LIN {X 0,Y 119.438,Z 237.503,A -85,B 0,C 180,E1 -30793.611,E2 -30793.611} C_VEL
LIN {X 0,Y 118.662,Z 241.868,A -85,B 0,C 180,E1 -30795.896,E2 -30795.896} C_VEL
LIN {X 0,Y 115.868,Z 252.745,A -85,B 0,C 180,E1 -30800.631,E2 -30800.631} C_VEL
LIN {X 0,Y 112.821,Z 263.888,A -85,B 0,C 180,E1 -30806.572,E2 -30806.572} C_VEL
LIN {X 0,Y 111.137,Z 271.247,A -85,B 0,C 180,E1 -30811.379,E2 -30811.379} C_VEL
LIN {X 0,Y 110.077,Z 278.124,A -85,B 0,C 180,E1 -30816.678,E2 -30816.678} C_VEL
LIN {X 0,Y 109.957,Z 285.411,A -85,B 0,C 180,E1 -30823.396,E2 -30823.396} C_VEL
LIN {X 0,Y 111.695,Z 292.264,A -85,B 0,C 180,E1 -30831.008,E2 -30831.008} C_VEL
LIN {X 0,Y 115.498,Z 297.926,A -85,B 0,C 180,E1 -30838.414,E2 -30838.414} C_VEL
LIN {X 0,Y 120.449,Z 301.979,A -85,B 0,C 180,E1 -30844.487,E2 -30844.487} C_VEL
LIN {X 0,Y 127.678,Z 305.592,A -85,B 0,C 180,E1 -30850.715,E2 -30850.715} C_VEL
LIN {X 0,Y 137.267,Z 308.443,A -85,B 0,C 180,E1 -30856.596,E2 -30856.596} C_VEL
LIN {X 0,Y 149.082,Z 310.385,A -85,B 0,C 180,E1 -30861.87,E2 -30861.87} C_VEL
LIN {X 0,Y 161.99,Z 311.348,A -85,B 0,C 180,E1 -30866.234,E2 -30866.234} C_VEL
LIN {X 0,Y 176.136,Z 311.421,A -85,B 0,C 180,E1 -30870,E2 -30870} C_VEL
LIN {X 0,Y 161.989,Z 311.349,A -85,B 0,C 180,E1 -30873.762,E2 -30873.762} C_VEL
LIN {X 0,Y 158.576,Z 311.223,A -85,B 0,C 180,E1 -30874.811,E2 -30874.811} C_VEL
LIN {X 0,Y 153.772,Z 311.084,A -85,B 0,C 180,E1 -30876.072,E2 -30876.072} C_VEL
LIN {X 0,Y 137.981,Z 310.516,A -85,B 0,C 180,E1 -30879.329,E2 -30879.329} C_VEL
LIN {X 0,Y 132.654,Z 310.062,A -85,B 0,C 180,E1 -30881.151,E2 -30881.151} C_VEL
LIN {X 0,Y 132.002,Z 309.878,A -85,B 0,C 180,E1 -30881.466,E2 -30881.466} C_VEL
LIN {X 0,Y 123.49,Z 307.999,A -85,B 0,C 180,E1 -30886.532,E2 -30886.532} C_VEL
LIN {X 0,Y 114.976,Z 304.68,A -85,B 0,C 180,E1 -30893.529,E2 -30893.529} C_VEL
LIN {X 0,Y 108.155,Z 299.529,A -85,B 0,C 180,E1 -30902.359,E2 -30902.359} C_VEL
LIN {X 0,Y 104.971,Z 294.579,A -85,B 0,C 180,E1 -30909.654,E2 -30909.654} C_VEL
LIN {X 0,Y 103.68,Z 288.412,A -85,B 0,C 180,E1 -30917.327,E2 -30917.327} C_VEL
LIN {X 0,Y 103.938,Z 283.545,A -85,B 0,C 180,E1 -30922.518,E2 -30922.518} C_VEL
LIN {X 0,Y 105.318,Z 276.622,A -85,B 0,C 180,E1 -30928.735,E2 -30928.735} C_VEL
LIN {X 0,Y 107.837,Z 268.159,A -85,B 0,C 180,E1 -30934.941,E2 -30934.941} C_VEL
LIN {X 0,Y 110.814,Z 259.529,A -85,B 0,C 180,E1 -30940.073,E2 -30940.073} C_VEL
LIN {X 0,Y 113.576,Z 251.659,A -85,B 0,C 180,E1 -30943.971,E2 -30943.971} C_VEL
LIN {X 0,Y 115.588,Z 245.687,A -85,B 0,C 180,E1 -30946.614,E2 -30946.614} C_VEL
LIN {X 0,Y 116.453,Z 242.049,A -85,B 0,C 180,E1 -30948.603,E2 -30948.603} C_VEL
LIN {X 0,Y 117.198,Z 238.265,A -85,B 0,C 180,E1 -30951.38,E2 -30951.38} C_VEL
LIN {X 0,Y 117.648,Z 235.676,A -85,B 0,C 180,E1 -30954.17,E2 -30954.17} C_VEL
LIN {X 0,Y 117.803,Z 234.235,A -85,B 0,C 180,E1 -30956.582,E2 -30956.582} C_VEL
LIN {X 0,Y 118.145,Z 232.807,A -85,B 0,C 180,E1 -30960.002,E2 -30960.002} C_VEL
LIN {X 0,Y 117.857,Z 233.676,A -85,B 0,C 180,E1 -30960.329,E2 -30960.329} C_VEL
LIN {X 0,Y 112.453,Z 246.435,A -85,B 0,C 180,E1 -30960.571,E2 -30960.571} C_VEL
LIN {X 0,Y 106.312,Z 257.337,A -85,B 0,C 180,E1 -30960.916,E2 -30960.916} C_VEL
LIN {X 0,Y 100.174,Z 266.275,A -85,B 0,C 180,E1 -30961.292,E2 -30961.292} C_VEL
LIN {X 0,Y 93.166,Z 274.795,A -85,B 0,C 180,E1 -30961.794,E2 -30961.794} C_VEL
LIN {X 0,Y 86.168,Z 282.007,A -85,B 0,C 180,E1 -30962.392,E2 -30962.392} C_VEL
LIN {X 0,Y 79.184,Z 288.203,A -85,B 0,C 180,E1 -30963.148,E2 -30963.148} C_VEL
LIN {X 0,Y 70.479,Z 294.736,A -85,B 0,C 180,E1 -30964.311,E2 -30964.311} C_VEL
LIN {X 0,Y 63.549,Z 299.237,A -85,B 0,C 180,E1 -30965.543,E2 -30965.543} C_VEL
LIN {X 0,Y 52.229,Z 305.189,A -85,B 0,C 180,E1 -30968.35,E2 -30968.35} C_VEL
LIN {X 0,Y 43.035,Z 309.057,A -85,B 0,C 180,E1 -30971.523,E2 -30971.523} C_VEL
LIN {X 0,Y 36.377,Z 311.428,A -85,B 0,C 180,E1 -30974.988,E2 -30974.988} C_VEL
LIN {X 0,Y 29.876,Z 313.231,A -85,B 0,C 180,E1 -30979.79,E2 -30979.79} C_VEL
LIN {X 0,Y 18.303,Z 315.698,A -85,B 0,C 180,E1 -30999.83,E2 -30999.83} C_VEL
LIN {X 0,Y 14.254,Z 316.299,A -85,B 0,C 180,E1 -31020.458,E2 -31020.458} C_VEL
LIN {X 0,Y 12.863,Z 316.464,A -85,B 0,C 180,E1 -31050,E2 -31050} C_VEL
LIN {X 0,Y 14.212,Z 316.298,A -85,B 0,C 180,E1 -31079.637,E2 -31079.637} C_VEL
LIN {X 0,Y 18.3,Z 315.698,A -85,B 0,C 180,E1 -31100.182,E2 -31100.182} C_VEL
LIN {X 0,Y 29.876,Z 313.231,A -85,B 0,C 180,E1 -31120.21,E2 -31120.21} C_VEL
LIN {X 0,Y 39.696,Z 310.276,A -85,B 0,C 180,E1 -31126.842,E2 -31126.842} C_VEL
LIN {X 0,Y 49.826,Z 306.286,A -85,B 0,C 180,E1 -31130.878,E2 -31130.878} C_VEL
LIN {X 0,Y 56.662,Z 303.07,A -85,B 0,C 180,E1 -31132.871,E2 -31132.871} C_VEL
LIN {X 0,Y 67.011,Z 297.047,A -85,B 0,C 180,E1 -31135.094,E2 -31135.094} C_VEL
LIN {X 0,Y 75.7,Z 290.954,A -85,B 0,C 180,E1 -31136.406,E2 -31136.406} C_VEL
LIN {X 0,Y 82.676,Z 285.259,A -85,B 0,C 180,E1 -31137.218,E2 -31137.218} C_VEL
LIN {X 0,Y 91.415,Z 276.712,A -85,B 0,C 180,E1 -31138.075,E2 -31138.075} C_VEL
LIN {X 0,Y 98.421,Z 268.542,A -85,B 0,C 180,E1 -31138.594,E2 -31138.594} C_VEL
LIN {X 0,Y 104.558,Z 260.038,A -85,B 0,C 180,E1 -31138.98,E2 -31138.98} C_VEL
LIN {X 0,Y 109.821,Z 251.33,A -85,B 0,C 180,E1 -31139.273,E2 -31139.273} C_VEL
LIN {X 0,Y 114.56,Z 241.781,A -85,B 0,C 180,E1 -31139.51,E2 -31139.51} C_VEL
LIN {X 0,Y 117.857,Z 233.673,A -85,B 0,C 180,E1 -31139.689,E2 -31139.689} C_VEL
LIN {X 0,Y 118.131,Z 232.849,A -85,B 0,C 180,E1 -31139.998,E2 -31139.998} C_VEL
LIN {X 0,Y 117.796,Z 234.256,A -85,B 0,C 180,E1 -31143.419,E2 -31143.419} C_VEL
LIN {X 0,Y 117.508,Z 236.547,A -85,B 0,C 180,E1 -31146.868,E2 -31146.868} C_VEL
LIN {X 0,Y 116.994,Z 239.333,A -85,B 0,C 180,E1 -31149.507,E2 -31149.507} C_VEL
LIN {X 0,Y 116.087,Z 243.786,A -85,B 0,C 180,E1 -31152.409,E2 -31152.409} C_VEL
LIN {X 0,Y 114.525,Z 248.785,A -85,B 0,C 180,E1 -31154.767,E2 -31154.767} C_VEL
LIN {X 0,Y 111.471,Z 257.668,A -85,B 0,C 180,E1 -31158.966,E2 -31158.966} C_VEL
LIN {X 0,Y 109.077,Z 264.504,A -85,B 0,C 180,E1 -31162.74,E2 -31162.74} C_VEL
LIN {X 0,Y 106.284,Z 272.99,A -85,B 0,C 180,E1 -31168.437,E2 -31168.437} C_VEL
LIN {X 0,Y 104.433,Z 280.285,A -85,B 0,C 180,E1 -31174.431,E2 -31174.431} C_VEL
LIN {X 0,Y 103.677,Z 286.441,A -85,B 0,C 180,E1 -31180.481,E2 -31180.481} C_VEL
LIN {X 0,Y 104.336,Z 292.655,A -85,B 0,C 180,E1 -31187.809,E2 -31187.809} C_VEL
LIN {X 0,Y 106.867,Z 298.01,A -85,B 0,C 180,E1 -31195.284,E2 -31195.284} C_VEL
LIN {X 0,Y 111.215,Z 302.267,A -85,B 0,C 180,E1 -31202.21,E2 -31202.21} C_VEL
LIN {X 0,Y 117.696,Z 305.878,A -85,B 0,C 180,E1 -31209.006,E2 -31209.006} C_VEL
LIN {X 0,Y 124.268,Z 308.213,A -85,B 0,C 180,E1 -31214.031,E2 -31214.031} C_VEL
LIN {X 0,Y 135.497,Z 310.434,A -85,B 0,C 180,E1 -31220.219,E2 -31220.219} C_VEL
LIN {X 0,Y 148.094,Z 311.583,A -85,B 0,C 180,E1 -31225.244,E2 -31225.244} C_VEL
LIN {X 0,Y 164.15,Z 311.737,A -85,B 0,C 180,E1 -31230,E2 -31230} C_VEL
LIN {X 0,Y 148.093,Z 311.584,A -85,B 0,C 180,E1 -31234.753,E2 -31234.753} C_VEL
LIN {X 0,Y 135.49,Z 310.441,A -85,B 0,C 180,E1 -31239.764,E2 -31239.764} C_VEL
LIN {X 0,Y 132.002,Z 309.878,A -85,B 0,C 180,E1 -31241.466,E2 -31241.466} C_VEL
LIN {X 0,Y 127.809,Z 309.35,A -85,B 0,C 180,E1 -31243.289,E2 -31243.289} C_VEL
LIN {X 0,Y 113.917,Z 307.957,A -85,B 0,C 180,E1 -31248.551,E2 -31248.551} C_VEL
LIN {X 0,Y 110.162,Z 307.095,A -85,B 0,C 180,E1 -31250.829,E2 -31250.829} C_VEL
LIN {X 0,Y 109.172,Z 306.728,A -85,B 0,C 180,E1 -31251.693,E2 -31251.693} C_VEL
LIN {X 0,Y 103.628,Z 303.627,A -85,B 0,C 180,E1 -31258.342,E2 -31258.342} C_VEL
LIN {X 0,Y 99.465,Z 299.348,A -85,B 0,C 180,E1 -31266.219,E2 -31266.219} C_VEL
LIN {X 0,Y 97.579,Z 294.398,A -85,B 0,C 180,E1 -31273.929,E2 -31273.929} C_VEL
LIN {X 0,Y 97.658,Z 287.855,A -85,B 0,C 180,E1 -31282.337,E2 -31282.337} C_VEL
LIN {X 0,Y 99.07,Z 282.136,A -85,B 0,C 180,E1 -31288.35,E2 -31288.35} C_VEL
LIN {X 0,Y 101.484,Z 275.444,A -85,B 0,C 180,E1 -31294.195,E2 -31294.195} C_VEL
LIN {X 0,Y 104.802,Z 267.508,A -85,B 0,C 180,E1 -31299.857,E2 -31299.857} C_VEL
LIN {X 0,Y 108.121,Z 259.958,A -85,B 0,C 180,E1 -31304.221,E2 -31304.221} C_VEL
LIN {X 0,Y 111.79,Z 251.291,A -85,B 0,C 180,E1 -31308.348,E2 -31308.348} C_VEL
LIN {X 0,Y 113.189,Z 247.517,A -85,B 0,C 180,E1 -31310.304,E2 -31310.304} C_VEL
LIN {X 0,Y 114.31,Z 243.924,A -85,B 0,C 180,E1 -31312.939,E2 -31312.939} C_VEL
LIN {X 0,Y 114.701,Z 242.248,A -85,B 0,C 180,E1 -31314.729,E2 -31314.729} C_VEL
LIN {X 0,Y 114.969,Z 241.111,A -85,B 0,C 180,E1 -31316.497,E2 -31316.497} C_VEL
LIN {X 0,Y 114.315,Z 242.512,A -85,B 0,C 180,E1 -31316.943,E2 -31316.943} C_VEL
LIN {X 0,Y 108.197,Z 254.379,A -85,B 0,C 180,E1 -31317.066,E2 -31317.066} C_VEL
LIN {X 0,Y 101.147,Z 264.951,A -85,B 0,C 180,E1 -31317.212,E2 -31317.212} C_VEL
LIN {X 0,Y 94.979,Z 272.687,A -85,B 0,C 180,E1 -31317.355,E2 -31317.355} C_VEL
LIN {X 0,Y 86.165,Z 281.815,A -85,B 0,C 180,E1 -31317.655,E2 -31317.655} C_VEL
LIN {X 0,Y 79.113,Z 288.012,A -85,B 0,C 180,E1 -31317.99,E2 -31317.99} C_VEL
LIN {X 0,Y 70.303,Z 294.545,A -85,B 0,C 180,E1 -31318.526,E2 -31318.526} C_VEL
LIN {X 0,Y 63.26,Z 299.045,A -85,B 0,C 180,E1 -31319.081,E2 -31319.081} C_VEL
LIN {X 0,Y 53.186,Z 304.328,A -85,B 0,C 180,E1 -31320.252,E2 -31320.252} C_VEL
LIN {X 0,Y 42.194,Z 308.865,A -85,B 0,C 180,E1 -31322.001,E2 -31322.001} C_VEL
LIN {X 0,Y 35.214,Z 311.237,A -85,B 0,C 180,E1 -31323.728,E2 -31323.728} C_VEL
LIN {X 0,Y 28.271,Z 313.04,A -85,B 0,C 180,E1 -31326.077,E2 -31326.077} C_VEL
LIN {X 0,Y 14.788,Z 315.507,A -85,B 0,C 180,E1 -31338.102,E2 -31338.102} C_VEL
LIN {X 0,Y 8.796,Z 316.109,A -85,B 0,C 180,E1 -31356.968,E2 -31356.968} C_VEL
LIN {X 0,Y 5.75,Z 316.273,A -85,B 0,C 180,E1 -31410,E2 -31410} C_VEL
LIN {X 0,Y 8.773,Z 316.108,A -85,B 0,C 180,E1 -31463.232,E2 -31463.232} C_VEL
LIN {X 0,Y 14.787,Z 315.507,A -85,B 0,C 180,E1 -31481.914,E2 -31481.914} C_VEL
LIN {X 0,Y 28.271,Z 313.04,A -85,B 0,C 180,E1 -31493.923,E2 -31493.923} C_VEL
LIN {X 0,Y 38.7,Z 310.085,A -85,B 0,C 180,E1 -31497.19,E2 -31497.19} C_VEL
LIN {X 0,Y 49.202,Z 306.095,A -85,B 0,C 180,E1 -31499.114,E2 -31499.114} C_VEL
LIN {X 0,Y 56.224,Z 302.878,A -85,B 0,C 180,E1 -31500.109,E2 -31500.109} C_VEL
LIN {X 0,Y 66.78,Z 296.856,A -85,B 0,C 180,E1 -31501.191,E2 -31501.191} C_VEL
LIN {X 0,Y 75.588,Z 290.762,A -85,B 0,C 180,E1 -31501.807,E2 -31501.807} C_VEL
LIN {X 0,Y 82.636,Z 285.068,A -85,B 0,C 180,E1 -31502.141,E2 -31502.141} C_VEL
LIN {X 0,Y 91.452,Z 276.521,A -85,B 0,C 180,E1 -31502.524,E2 -31502.524} C_VEL
LIN {X 0,Y 98.503,Z 268.351,A -85,B 0,C 180,E1 -31502.724,E2 -31502.724} C_VEL
LIN {X 0,Y 104.673,Z 259.847,A -85,B 0,C 180,E1 -31502.872,E2 -31502.872} C_VEL
LIN {X 0,Y 110.366,Z 250.392,A -85,B 0,C 180,E1 -31503.004,E2 -31503.004} C_VEL
LIN {X 0,Y 114.153,Z 242.882,A -85,B 0,C 180,E1 -31503.048,E2 -31503.048} C_VEL
LIN {X 0,Y 114.958,Z 241.136,A -85,B 0,C 180,E1 -31503.503,E2 -31503.503} C_VEL
LIN {X 0,Y 114.708,Z 242.232,A -85,B 0,C 180,E1 -31505.271,E2 -31505.271} C_VEL
LIN {X 0,Y 114.078,Z 244.695,A -85,B 0,C 180,E1 -31507.642,E2 -31507.642} C_VEL
LIN {X 0,Y 113.171,Z 247.553,A -85,B 0,C 180,E1 -31509.699,E2 -31509.699} C_VEL
LIN {X 0,Y 111.781,Z 251.303,A -85,B 0,C 180,E1 -31511.648,E2 -31511.648} C_VEL
LIN {X 0,Y 107.546,Z 261.415,A -85,B 0,C 180,E1 -31516.579,E2 -31516.579} C_VEL
LIN {X 0,Y 102.944,Z 271.932,A -85,B 0,C 180,E1 -31523.11,E2 -31523.11} C_VEL
LIN {X 0,Y 99.555,Z 280.572,A -85,B 0,C 180,E1 -31530.147,E2 -31530.147} C_VEL
LIN {X 0,Y 97.91,Z 286.701,A -85,B 0,C 180,E1 -31536.364,E2 -31536.364} C_VEL
LIN {X 0,Y 97.409,Z 292.784,A -85,B 0,C 180,E1 -31543.823,E2 -31543.823} C_VEL
LIN {X 0,Y 98.744,Z 297.982,A -85,B 0,C 180,E1 -31551.524,E2 -31551.524} C_VEL
LIN {X 0,Y 102.104,Z 302.412,A -85,B 0,C 180,E1 -31559.271,E2 -31559.271} C_VEL
LIN {X 0,Y 107.87,Z 306.162,A -85,B 0,C 180,E1 -31566.989,E2 -31566.989} C_VEL
LIN {X 0,Y 113.189,Z 308.289,A -85,B 0,C 180,E1 -31571.914,E2 -31571.914} C_VEL
LIN {X 0,Y 122.122,Z 310.418,A -85,B 0,C 180,E1 -31578.042,E2 -31578.042} C_VEL
LIN {X 0,Y 134.394,Z 311.803,A -85,B 0,C 180,E1 -31583.997,E2 -31583.997} C_VEL
LIN {X 0,Y 147.624,Z 312.173,A -85,B 0,C 180,E1 -31588.66,E2 -31588.66} C_VEL
LIN {X 0,Y 152.223,Z 312.051,A -85,B 0,C 180,E1 -31590,E2 -31590} C_VEL
LIN {X 0,Y 140.825,Z 312.065,A -85,B 0,C 180,E1 -31593.543,E2 -31593.543} C_VEL
LIN {X 0,Y 128.009,Z 311.191,A -85,B 0,C 180,E1 -31598.806,E2 -31598.806} C_VEL
LIN {X 0,Y 119.334,Z 309.848,A -85,B 0,C 180,E1 -31603.625,E2 -31603.625} C_VEL
LIN {X 0,Y 111.719,Z 307.776,A -85,B 0,C 180,E1 -31609.338,E2 -31609.338} C_VEL
LIN {X 0,Y 109.172,Z 306.728,A -85,B 0,C 180,E1 -31611.693,E2 -31611.693} C_VEL
LIN {X 0,Y 106.013,Z 305.743,A -85,B 0,C 180,E1 -31614.302,E2 -31614.302} C_VEL
LIN {X 0,Y 95.36,Z 303.145,A -85,B 0,C 180,E1 -31622.33,E2 -31622.33} C_VEL
LIN {X 0,Y 92.785,Z 301.661,A -85,B 0,C 180,E1 -31626.088,E2 -31626.088} C_VEL
LIN {X 0,Y 92.582,Z 301.332,A -85,B 0,C 180,E1 -31626.657,E2 -31626.657} C_VEL
LIN {X 0,Y 90.988,Z 296.082,A -85,B 0,C 180,E1 -31635.963,E2 -31635.963} C_VEL
LIN {X 0,Y 91.838,Z 289.677,A -85,B 0,C 180,E1 -31644.98,E2 -31644.98} C_VEL
LIN {X 0,Y 94.652,Z 282.378,A -85,B 0,C 180,E1 -31653,E2 -31653} C_VEL
LIN {X 0,Y 98.048,Z 275.499,A -85,B 0,C 180,E1 -31659.001,E2 -31659.001} C_VEL
LIN {X 0,Y 101.83,Z 268.389,A -85,B 0,C 180,E1 -31663.977,E2 -31663.977} C_VEL
LIN {X 0,Y 106.055,Z 260.347,A -85,B 0,C 180,E1 -31668.535,E2 -31668.535} C_VEL
LIN {X 0,Y 109.351,Z 253.877,A -85,B 0,C 180,E1 -31671.616,E2 -31671.616} C_VEL
LIN {X 0,Y 110.135,Z 251.985,A -85,B 0,C 180,E1 -31672.67,E2 -31672.67} C_VEL
LIN {X 0,Y 109.077,Z 253.677,A -85,B 0,C 180,E1 -31673.347,E2 -31673.347} C_VEL
LIN {X 0,Y 101.741,Z 264.76,A -85,B 0,C 180,E1 -31673.207,E2 -31673.207} C_VEL
LIN {X 0,Y 95.568,Z 272.496,A -85,B 0,C 180,E1 -31673.107,E2 -31673.107} C_VEL
LIN {X 0,Y 86.75,Z 281.624,A -85,B 0,C 180,E1 -31672.94,E2 -31672.94} C_VEL
LIN {X 0,Y 79.683,Z 287.821,A -85,B 0,C 180,E1 -31672.859,E2 -31672.859} C_VEL
LIN {X 0,Y 70.846,Z 294.353,A -85,B 0,C 180,E1 -31672.75,E2 -31672.75} C_VEL
LIN {X 0,Y 63.775,Z 298.853,A -85,B 0,C 180,E1 -31672.658,E2 -31672.658} C_VEL
LIN {X 0,Y 52.639,Z 304.573,A -85,B 0,C 180,E1 -31672.585,E2 -31672.585} C_VEL
LIN {X 0,Y 42.544,Z 308.674,A -85,B 0,C 180,E1 -31672.375,E2 -31672.375} C_VEL
LIN {X 0,Y 35.47,Z 311.046,A -85,B 0,C 180,E1 -31672.177,E2 -31672.177} C_VEL
LIN {X 0,Y 28.413,Z 312.849,A -85,B 0,C 180,E1 -31671.655,E2 -31671.655} C_VEL
LIN {X 0,Y 14.285,Z 315.315,A -85,B 0,C 180,E1 -31669.716,E2 -31669.716} C_VEL
LIN {X 0,Y 7.266,Z 315.917,A -85,B 0,C 180,E1 -31665.308,E2 -31665.308} C_VEL
LIN {X 0,Y 1.349,Z 316.083,A -85,B 0,C 180,E1 -31590,E2 -31590} C_VEL
LIN {X 0,Y 7.274,Z 315.916,A -85,B 0,C 180,E1 -31514.942,E2 -31514.942} C_VEL
LIN {X 0,Y 14.286,Z 315.315,A -85,B 0,C 180,E1 -31510.299,E2 -31510.299} C_VEL
LIN {X 0,Y 28.413,Z 312.849,A -85,B 0,C 180,E1 -31508.345,E2 -31508.345} C_VEL
LIN {X 0,Y 39.009,Z 309.893,A -85,B 0,C 180,E1 -31507.738,E2 -31507.738} C_VEL
LIN {X 0,Y 49.608,Z 305.903,A -85,B 0,C 180,E1 -31507.387,E2 -31507.387} C_VEL
LIN {X 0,Y 56.687,Z 302.687,A -85,B 0,C 180,E1 -31507.326,E2 -31507.326} C_VEL
LIN {X 0,Y 67.307,Z 296.664,A -85,B 0,C 180,E1 -31507.269,E2 -31507.269} C_VEL
LIN {X 0,Y 76.146,Z 290.571,A -85,B 0,C 180,E1 -31507.168,E2 -31507.168} C_VEL
LIN {X 0,Y 83.205,Z 284.878,A -85,B 0,C 180,E1 -31507.037,E2 -31507.037} C_VEL
LIN {X 0,Y 92.039,Z 276.331,A -85,B 0,C 180,E1 -31506.943,E2 -31506.943} C_VEL
LIN {X 0,Y 99.094,Z 268.161,A -85,B 0,C 180,E1 -31506.825,E2 -31506.825} C_VEL
LIN {X 0,Y 105.268,Z 259.657,A -85,B 0,C 180,E1 -31506.736,E2 -31506.736} C_VEL
LIN {X 0,Y 109.067,Z 253.699,A -85,B 0,C 180,E1 -31506.666,E2 -31506.666} C_VEL
LIN {X 0,Y 110.122,Z 252.009,A -85,B 0,C 180,E1 -31507.331,E2 -31507.331} C_VEL
LIN {X 0,Y 108.665,Z 255.267,A -85,B 0,C 180,E1 -31509.027,E2 -31509.027} C_VEL
LIN {X 0,Y 103.864,Z 264.619,A -85,B 0,C 180,E1 -31513.787,E2 -31513.787} C_VEL
LIN {X 0,Y 99.091,Z 273.519,A -85,B 0,C 180,E1 -31519.503,E2 -31519.503} C_VEL
LIN {X 0,Y 95.367,Z 280.812,A -85,B 0,C 180,E1 -31525.483,E2 -31525.483} C_VEL
LIN {X 0,Y 92.664,Z 287.185,A -85,B 0,C 180,E1 -31532.064,E2 -31532.064} C_VEL
LIN {X 0,Y 91.097,Z 293.038,A -85,B 0,C 180,E1 -31539.513,E2 -31539.513} C_VEL
LIN {X 0,Y 91.269,Z 298.126,A -85,B 0,C 180,E1 -31547.495,E2 -31547.495} C_VEL
LIN {X 0,Y 93.441,Z 302.552,A -85,B 0,C 180,E1 -31555.822,E2 -31555.822} C_VEL
LIN {X 0,Y 98.426,Z 306.44,A -85,B 0,C 180,E1 -31564.633,E2 -31564.633} C_VEL
LIN {X 0,Y 104.076,Z 308.843,A -85,B 0,C 180,E1 -31570.97,E2 -31570.97} C_VEL
LIN {X 0,Y 114.568,Z 311.171,A -85,B 0,C 180,E1 -31578.95,E2 -31578.95} C_VEL
LIN {X 0,Y 123.013,Z 312.105,A -85,B 0,C 180,E1 -31583.439,E2 -31583.439} C_VEL
LIN {X 0,Y 133.631,Z 312.512,A -85,B 0,C 180,E1 -31587.747,E2 -31587.747} C_VEL
LIN {X 0,Y 140.339,Z 312.363,A -85,B 0,C 180,E1 -31590,E2 -31590} C_VEL
LIN {X 0,Y 126.948,Z 312.274,A -85,B 0,C 180,E1 -31594.816,E2 -31594.816} C_VEL
LIN {X 0,Y 120.567,Z 311.94,A -85,B 0,C 180,E1 -31597.728,E2 -31597.728} C_VEL
LIN {X 0,Y 108.903,Z 310.136,A -85,B 0,C 180,E1 -31604.96,E2 -31604.96} C_VEL
LIN {X 0,Y 102.954,Z 308.495,A -85,B 0,C 180,E1 -31610.112,E2 -31610.112} C_VEL
LIN {X 0,Y 96.203,Z 305.083,A -85,B 0,C 180,E1 -31618.765,E2 -31618.765} C_VEL
LIN {X 0,Y 92.582,Z 301.332,A -85,B 0,C 180,E1 -31626.657,E2 -31626.657} C_VEL
LIN {X 0,Y 91.075,Z 299.812,A -85,B 0,C 180,E1 -31630.099,E2 -31630.099} C_VEL
LIN {X 0,Y 85.684,Z 295.681,A -85,B 0,C 180,E1 -31640.809,E2 -31640.809} C_VEL
LIN {X 0,Y 85.348,Z 293.771,A -85,B 0,C 180,E1 -31644.529,E2 -31644.529} C_VEL
LIN {X 0,Y 85.568,Z 293.016,A -85,B 0,C 180,E1 -31645.732,E2 -31645.732} C_VEL
LIN {X 0,Y 89.351,Z 285.459,A -85,B 0,C 180,E1 -31655.21,E2 -31655.21} C_VEL
LIN {X 0,Y 94.253,Z 277.399,A -85,B 0,C 180,E1 -31662.649,E2 -31662.649} C_VEL
LIN {X 0,Y 99.429,Z 269.253,A -85,B 0,C 180,E1 -31668.318,E2 -31668.318} C_VEL
LIN {X 0,Y 100.183,Z 267.971,A -85,B 0,C 180,E1 -31669.148,E2 -31669.148} C_VEL
LIN {X 0,Y 93.173,Z 276.139,A -85,B 0,C 180,E1 -31668.689,E2 -31668.689} C_VEL
LIN {X 0,Y 84.389,Z 284.685,A -85,B 0,C 180,E1 -31668.11,E2 -31668.11} C_VEL
LIN {X 0,Y 73.844,Z 293.008,A -85,B 0,C 180,E1 -31667.298,E2 -31667.298} C_VEL
LIN {X 0,Y 65.072,Z 298.662,A -85,B 0,C 180,E1 -31666.416,E2 -31666.416} C_VEL
LIN {X 0,Y 55.039,Z 303.932,A -85,B 0,C 180,E1 -31665.208,E2 -31665.208} C_VEL
LIN {X 0,Y 47.521,Z 307.244,A -85,B 0,C 180,E1 -31664.006,E2 -31664.006} C_VEL
LIN {X 0,Y 37.122,Z 310.855,A -85,B 0,C 180,E1 -31661.194,E2 -31661.194} C_VEL
LIN {X 0,Y 23.552,Z 314.053,A -85,B 0,C 180,E1 -31653.536,E2 -31653.536} C_VEL
LIN {X 0,Y 17.071,Z 315.124,A -85,B 0,C 180,E1 -31645.424,E2 -31645.424} C_VEL
LIN {X 0,Y 11.393,Z 315.726,A -85,B 0,C 180,E1 -31628.089,E2 -31628.089} C_VEL
LIN {X 0,Y 8.44,Z 315.892,A -85,B 0,C 180,E1 -31590,E2 -31590} C_VEL
LIN {X 0,Y 11.414,Z 315.725,A -85,B 0,C 180,E1 -31551.993,E2 -31551.993} C_VEL
LIN {X 0,Y 17.073,Z 315.124,A -85,B 0,C 180,E1 -31534.585,E2 -31534.585} C_VEL
LIN {X 0,Y 30.274,Z 312.658,A -85,B 0,C 180,E1 -31521.784,E2 -31521.784} C_VEL
LIN {X 0,Y 40.592,Z 309.701,A -85,B 0,C 180,E1 -31517.779,E2 -31517.779} C_VEL
LIN {X 0,Y 51.024,Z 305.711,A -85,B 0,C 180,E1 -31515.384,E2 -31515.384} C_VEL
LIN {X 0,Y 61.543,Z 300.579,A -85,B 0,C 180,E1 -31513.914,E2 -31513.914} C_VEL
LIN {X 0,Y 70.329,Z 295.318,A -85,B 0,C 180,E1 -31513.013,E2 -31513.013} C_VEL
LIN {X 0,Y 79.113,Z 289.006,A -85,B 0,C 180,E1 -31512.265,E2 -31512.265} C_VEL
LIN {X 0,Y 86.139,Z 283.06,A -85,B 0,C 180,E1 -31511.743,E2 -31511.743} C_VEL
LIN {X 0,Y 93.165,Z 276.14,A -85,B 0,C 180,E1 -31511.285,E2 -31511.285} C_VEL
LIN {X 0,Y 100.189,Z 267.97,A -85,B 0,C 180,E1 -31510.868,E2 -31510.868} C_VEL
LIN {X 0,Y 95.153,Z 275.916,A -85,B 0,C 180,E1 -31516.225,E2 -31516.225} C_VEL
LIN {X 0,Y 90.375,Z 283.575,A -85,B 0,C 180,E1 -31522.879,E2 -31522.879} C_VEL
LIN {X 0,Y 86.366,Z 291.223,A -85,B 0,C 180,E1 -31531.711,E2 -31531.711} C_VEL
LIN {X 0,Y 84.488,Z 297.663,A -85,B 0,C 180,E1 -31541.715,E2 -31541.715} C_VEL
LIN {X 0,Y 85.32,Z 302.555,A -85,B 0,C 180,E1 -31551.486,E2 -31551.486} C_VEL
LIN {X 0,Y 88.655,Z 306.327,A -85,B 0,C 180,E1 -31560.688,E2 -31560.688} C_VEL
LIN {X 0,Y 93.375,Z 308.855,A -85,B 0,C 180,E1 -31567.893,E2 -31567.893} C_VEL
LIN {X 0,Y 101.453,Z 311.082,A -85,B 0,C 180,E1 -31575.88,E2 -31575.88} C_VEL
LIN {X 0,Y 113.182,Z 312.462,A -85,B 0,C 180,E1 -31583.453,E2 -31583.453} C_VEL
LIN {X 0,Y 126.512,Z 312.728,A -85,B 0,C 180,E1 -31589.213,E2 -31589.213} C_VEL
LIN {X 0,Y 128.675,Z 312.67,A -85,B 0,C 180,E1 -31590,E2 -31590} C_VEL
LIN {X 0,Y 119.689,Z 312.746,A -85,B 0,C 180,E1 -31593.451,E2 -31593.451} C_VEL
LIN {X 0,Y 107.07,Z 311.897,A -85,B 0,C 180,E1 -31600.083,E2 -31600.083} C_VEL
LIN {X 0,Y 98.634,Z 310.423,A -85,B 0,C 180,E1 -31606.56,E2 -31606.56} C_VEL
LIN {X 0,Y 92.129,Z 308.307,A -85,B 0,C 180,E1 -31613.742,E2 -31613.742} C_VEL
LIN {X 0,Y 86.359,Z 304.17,A -85,B 0,C 180,E1 -31624.727,E2 -31624.727} C_VEL
LIN {X 0,Y 84.431,Z 299.411,A -85,B 0,C 180,E1 -31634.969,E2 -31634.969} C_VEL
LIN {X 0,Y 85.338,Z 293.631,A -85,B 0,C 180,E1 -31644.8,E2 -31644.8} C_VEL
LIN {X 0,Y 85.568,Z 293.016,A -85,B 0,C 180,E1 -31645.732,E2 -31645.732} C_VEL
LIN {X 0,Y 85.701,Z 291.667,A -85,B 0,C 180,E1 -31648.248,E2 -31648.248} C_VEL
LIN {X 0,Y 84.312,Z 288.345,A -85,B 0,C 180,E1 -31657.034,E2 -31657.034} C_VEL
LIN {X 0,Y 85.178,Z 286.754,A -85,B 0,C 180,E1 -31659.423,E2 -31659.423} C_VEL
LIN {X 0,Y 88.012,Z 282.855,A -85,B 0,C 180,E1 -31663.381,E2 -31663.381} C_VEL
LIN {X 0,Y 87.887,Z 282.867,A -85,B 0,C 180,E1 -31663.657,E2 -31663.657} C_VEL
LIN {X 0,Y 80.932,Z 288.814,A -85,B 0,C 180,E1 -31662.788,E2 -31662.788} C_VEL
LIN {X 0,Y 72.277,Z 295.126,A -85,B 0,C 180,E1 -31661.451,E2 -31661.451} C_VEL
LIN {X 0,Y 63.647,Z 300.387,A -85,B 0,C 180,E1 -31659.813,E2 -31659.813} C_VEL
LIN {X 0,Y 53.371,Z 305.519,A -85,B 0,C 180,E1 -31657.187,E2 -31657.187} C_VEL
LIN {X 0,Y 43.307,Z 309.51,A -85,B 0,C 180,E1 -31653.196,E2 -31653.196} C_VEL
LIN {X 0,Y 33.568,Z 312.467,A -85,B 0,C 180,E1 -31646.873,E2 -31646.873} C_VEL
LIN {X 0,Y 21.918,Z 314.932,A -85,B 0,C 180,E1 -31629.889,E2 -31629.889} C_VEL
LIN {X 0,Y 17.55,Z 315.535,A -85,B 0,C 180,E1 -31613.606,E2 -31613.606} C_VEL
LIN {X 0,Y 15.549,Z 315.702,A -85,B 0,C 180,E1 -31590,E2 -31590} C_VEL
LIN {X 0,Y 17.57,Z 315.535,A -85,B 0,C 180,E1 -31566.422,E2 -31566.422} C_VEL
LIN {X 0,Y 21.92,Z 314.932,A -85,B 0,C 180,E1 -31550.115,E2 -31550.115} C_VEL
LIN {X 0,Y 33.568,Z 312.467,A -85,B 0,C 180,E1 -31533.127,E2 -31533.127} C_VEL
LIN {X 0,Y 43.306,Z 309.51,A -85,B 0,C 180,E1 -31526.802,E2 -31526.802} C_VEL
LIN {X 0,Y 53.365,Z 305.52,A -85,B 0,C 180,E1 -31522.797,E2 -31522.797} C_VEL
LIN {X 0,Y 63.64,Z 300.388,A -85,B 0,C 180,E1 -31520.168,E2 -31520.168} C_VEL
LIN {X 0,Y 72.271,Z 295.127,A -85,B 0,C 180,E1 -31518.535,E2 -31518.535} C_VEL
LIN {X 0,Y 80.923,Z 288.815,A -85,B 0,C 180,E1 -31517.191,E2 -31517.191} C_VEL
LIN {X 0,Y 87.862,Z 282.869,A -85,B 0,C 180,E1 -31516.289,E2 -31516.289} C_VEL
LIN {X 0,Y 88.004,Z 282.856,A -85,B 0,C 180,E1 -31516.601,E2 -31516.601} C_VEL
LIN {X 0,Y 83.792,Z 288.589,A -85,B 0,C 180,E1 -31522.689,E2 -31522.689} C_VEL
LIN {X 0,Y 79.658,Z 295.226,A -85,B 0,C 180,E1 -31531.959,E2 -31531.959} C_VEL
LIN {X 0,Y 77.9,Z 300.288,A -85,B 0,C 180,E1 -31541.37,E2 -31541.37} C_VEL
LIN {X 0,Y 78.904,Z 305.265,A -85,B 0,C 180,E1 -31553.282,E2 -31553.282} C_VEL
LIN {X 0,Y 84.508,Z 309.356,A -85,B 0,C 180,E1 -31566.171,E2 -31566.171} C_VEL
LIN {X 0,Y 93.874,Z 311.8,A -85,B 0,C 180,E1 -31576.71,E2 -31576.71} C_VEL
LIN {X 0,Y 101.062,Z 312.698,A -85,B 0,C 180,E1 -31582.005,E2 -31582.005} C_VEL
LIN {X 0,Y 112.509,Z 313.102,A -85,B 0,C 180,E1 -31588.054,E2 -31588.054} C_VEL
LIN {X 0,Y 117.175,Z 312.975,A -85,B 0,C 180,E1 -31590,E2 -31590} C_VEL
LIN {X 0,Y 105.846,Z 312.931,A -85,B 0,C 180,E1 -31595.165,E2 -31595.165} C_VEL
LIN {X 0,Y 99.604,Z 312.602,A -85,B 0,C 180,E1 -31598.962,E2 -31598.962} C_VEL
LIN {X 0,Y 88.552,Z 310.706,A -85,B 0,C 180,E1 -31608.509,E2 -31608.509} C_VEL
LIN {X 0,Y 83.975,Z 309.129,A -85,B 0,C 180,E1 -31614.737,E2 -31614.737} C_VEL
LIN {X 0,Y 78.889,Z 305.276,A -85,B 0,C 180,E1 -31626.704,E2 -31626.704} C_VEL
LIN {X 0,Y 77.879,Z 300.299,A -85,B 0,C 180,E1 -31638.625,E2 -31638.625} C_VEL
LIN {X 0,Y 79.634,Z 295.244,A -85,B 0,C 180,E1 -31648.03,E2 -31648.03} C_VEL
LIN {X 0,Y 83.067,Z 289.642,A -85,B 0,C 180,E1 -31656.04,E2 -31656.04} C_VEL
LIN {X 0,Y 85.178,Z 286.754,A -85,B 0,C 180,E1 -31659.423,E2 -31659.423} C_VEL
LIN {X 0,Y 83.974,Z 287.733,A -85,B 0,C 180,E1 -31659.304,E2 -31659.304} C_VEL
LIN {X 0,Y 80.616,Z 291.046,A -85,B 0,C 180,E1 -31657.082,E2 -31657.082} C_VEL
LIN {X 0,Y 74.549,Z 297.408,A -85,B 0,C 180,E1 -31649.766,E2 -31649.766} C_VEL
LIN {X 0,Y 71.99,Z 300.771,A -85,B 0,C 180,E1 -31643.87,E2 -31643.87} C_VEL
LIN {X 0,Y 71.551,Z 301.718,A -85,B 0,C 180,E1 -31641.726,E2 -31641.726} C_VEL
LIN {X 0,Y 71.664,Z 306.536,A -85,B 0,C 180,E1 -31628.326,E2 -31628.326} C_VEL
LIN {X 0,Y 74.811,Z 309.404,A -85,B 0,C 180,E1 -31618.016,E2 -31618.016} C_VEL
LIN {X 0,Y 81.169,Z 311.648,A -85,B 0,C 180,E1 -31607.752,E2 -31607.752} C_VEL
LIN {X 0,Y 92.179,Z 313.081,A -85,B 0,C 180,E1 -31597.643,E2 -31597.643} C_VEL
LIN {X 0,Y 98.586,Z 313.392,A -85,B 0,C 180,E1 -31593.63,E2 -31593.63} C_VEL
LIN {X 0,Y 105.908,Z 313.277,A -85,B 0,C 180,E1 -31590,E2 -31590} C_VEL
LIN {X 0,Y 97.707,Z 313.352,A -85,B 0,C 180,E1 -31585.875,E2 -31585.875} C_VEL
LIN {X 0,Y 86.324,Z 312.514,A -85,B 0,C 180,E1 -31577.668,E2 -31577.668} C_VEL
LIN {X 0,Y 78.82,Z 310.984,A -85,B 0,C 180,E1 -31569.105,E2 -31569.105} C_VEL
LIN {X 0,Y 73.65,Z 308.652,A -85,B 0,C 180,E1 -31559.178,E2 -31559.178} C_VEL
LIN {X 0,Y 71.125,Z 304.696,A -85,B 0,C 180,E1 -31546.237,E2 -31546.237} C_VEL
LIN {X 0,Y 71.934,Z 300.634,A -85,B 0,C 180,E1 -31535.884,E2 -31535.884} C_VEL
LIN {X 0,Y 74.272,Z 296.821,A -85,B 0,C 180,E1 -31528.234,E2 -31528.234} C_VEL
LIN {X 0,Y 76.077,Z 294.316,A -85,B 0,C 180,E1 -31524.131,E2 -31524.131} C_VEL
LIN {X 0,Y 73.151,Z 296.091,A -85,B 0,C 180,E1 -31524.117,E2 -31524.117} C_VEL
LIN {X 0,Y 63.1,Z 302.112,A -85,B 0,C 180,E1 -31526.998,E2 -31526.998} C_VEL
LIN {X 0,Y 53.255,Z 306.861,A -85,B 0,C 180,E1 -31530.929,E2 -31530.929} C_VEL
LIN {X 0,Y 43.87,Z 310.471,A -85,B 0,C 180,E1 -31536.775,E2 -31536.775} C_VEL
LIN {X 0,Y 37.943,Z 312.276,A -85,B 0,C 180,E1 -31542.192,E2 -31542.192} C_VEL
LIN {X 0,Y 27.762,Z 314.741,A -85,B 0,C 180,E1 -31559.582,E2 -31559.582} C_VEL
LIN {X 0,Y 24.275,Z 315.343,A -85,B 0,C 180,E1 -31573.171,E2 -31573.171} C_VEL
LIN {X 0,Y 22.647,Z 315.511,A -85,B 0,C 180,E1 -31590,E2 -31590} C_VEL
LIN {X 0,Y 24.258,Z 315.344,A -85,B 0,C 180,E1 -31606.841,E2 -31606.841} C_VEL
LIN {X 0,Y 27.761,Z 314.741,A -85,B 0,C 180,E1 -31620.42,E2 -31620.42} C_VEL
LIN {X 0,Y 37.943,Z 312.276,A -85,B 0,C 180,E1 -31637.808,E2 -31637.808} C_VEL
LIN {X 0,Y 46.952,Z 309.319,A -85,B 0,C 180,E1 -31645.412,E2 -31645.412} C_VEL
LIN {X 0,Y 56.524,Z 305.328,A -85,B 0,C 180,E1 -31650.499,E2 -31650.499} C_VEL
LIN {X 0,Y 66.455,Z 300.195,A -85,B 0,C 180,E1 -31654.016,E2 -31654.016} C_VEL
LIN {X 0,Y 73.161,Z 296.09,A -85,B 0,C 180,E1 -31655.865,E2 -31655.865} C_VEL
LIN {X 0,Y 76.097,Z 294.307,A -85,B 0,C 180,E1 -31655.858,E2 -31655.858} C_VEL
LIN {X 0,Y 72.443,Z 299.605,A -85,B 0,C 180,E1 -31646.315,E2 -31646.315} C_VEL
LIN {X 0,Y 71.551,Z 301.718,A -85,B 0,C 180,E1 -31641.726,E2 -31641.726} C_VEL
LIN {X 0,Y 70.499,Z 303.679,A -85,B 0,C 180,E1 -31637.292,E2 -31637.292} C_VEL
LIN {X 0,Y 68.023,Z 306.954,A -85,B 0,C 180,E1 -31629.79,E2 -31629.79} C_VEL
LIN {X 0,Y 66.898,Z 309.625,A -85,B 0,C 180,E1 -31621.781,E2 -31621.781} C_VEL
LIN {X 0,Y 67.959,Z 310.647,A -85,B 0,C 180,E1 -31616.973,E2 -31616.973} C_VEL
LIN {X 0,Y 73.99,Z 312.432,A -85,B 0,C 180,E1 -31606.556,E2 -31606.556} C_VEL
LIN {X 0,Y 79.954,Z 313.272,A -85,B 0,C 180,E1 -31600.125,E2 -31600.125} C_VEL
LIN {X 0,Y 91.407,Z 313.668,A -85,B 0,C 180,E1 -31591.845,E2 -31591.845} C_VEL
LIN {X 0,Y 94.825,Z 313.575,A -85,B 0,C 180,E1 -31590,E2 -31590} C_VEL
LIN {X 0,Y 84.811,Z 313.54,A -85,B 0,C 180,E1 -31583.905,E2 -31583.905} C_VEL
LIN {X 0,Y 78.796,Z 313.198,A -85,B 0,C 180,E1 -31578.833,E2 -31578.833} C_VEL
LIN {X 0,Y 69.266,Z 311.23,A -85,B 0,C 180,E1 -31565.939,E2 -31565.939} C_VEL
LIN {X 0,Y 65.167,Z 308.685,A -85,B 0,C 180,E1 -31553.819,E2 -31553.819} C_VEL
LIN {X 0,Y 64.484,Z 305.121,A -85,B 0,C 180,E1 -31540.834,E2 -31540.834} C_VEL
LIN {X 0,Y 65.551,Z 302.866,A -85,B 0,C 180,E1 -31534.144,E2 -31534.144} C_VEL
LIN {X 0,Y 61.747,Z 304.438,A -85,B 0,C 180,E1 -31534.683,E2 -31534.683} C_VEL
LIN {X 0,Y 54.229,Z 307.911,A -85,B 0,C 180,E1 -31538.96,E2 -31538.96} C_VEL
LIN {X 0,Y 48.485,Z 310.279,A -85,B 0,C 180,E1 -31543.551,E2 -31543.551} C_VEL
LIN {X 0,Y 43.06,Z 312.084,A -85,B 0,C 180,E1 -31549.243,E2 -31549.243} C_VEL
LIN {X 0,Y 34.108,Z 314.55,A -85,B 0,C 180,E1 -31565.663,E2 -31565.663} C_VEL
LIN {X 0,Y 31.16,Z 315.152,A -85,B 0,C 180,E1 -31576.965,E2 -31576.965} C_VEL
LIN {X 0,Y 29.762,Z 315.32,A -85,B 0,C 180,E1 -31590,E2 -31590} C_VEL
LIN {X 0,Y 31.146,Z 315.153,A -85,B 0,C 180,E1 -31603.041,E2 -31603.041} C_VEL
LIN {X 0,Y 34.106,Z 314.55,A -85,B 0,C 180,E1 -31614.338,E2 -31614.338} C_VEL
LIN {X 0,Y 43.06,Z 312.084,A -85,B 0,C 180,E1 -31630.757,E2 -31630.757} C_VEL
LIN {X 0,Y 51.329,Z 309.128,A -85,B 0,C 180,E1 -31638.856,E2 -31638.856} C_VEL
LIN {X 0,Y 60.363,Z 305.136,A -85,B 0,C 180,E1 -31644.587,E2 -31644.587} C_VEL
LIN {X 0,Y 61.391,Z 304.628,A -85,B 0,C 180,E1 -31645.087,E2 -31645.087} C_VEL
LIN {X 0,Y 65.558,Z 302.862,A -85,B 0,C 180,E1 -31645.862,E2 -31645.862} C_VEL
LIN {X 0,Y 64.319,Z 306.454,A -85,B 0,C 180,E1 -31634.995,E2 -31634.995} C_VEL
LIN {X 0,Y 66.19,Z 309.721,A -85,B 0,C 180,E1 -31621.856,E2 -31621.856} C_VEL
LIN {X 0,Y 67.959,Z 310.647,A -85,B 0,C 180,E1 -31616.973,E2 -31616.973} C_VEL
LIN {X 0,Y 69.532,Z 311.673,A -85,B 0,C 180,E1 -31612.279,E2 -31612.279} C_VEL
LIN {X 0,Y 71.537,Z 313.016,A -85,B 0,C 180,E1 -31604.451,E2 -31604.451} C_VEL
LIN {X 0,Y 74.898,Z 313.868,A -85,B 0,C 180,E1 -31597.205,E2 -31597.205} C_VEL
LIN {X 0,Y 78.383,Z 313.972,A -85,B 0,C 180,E1 -31593.663,E2 -31593.663} C_VEL
LIN {X 0,Y 83.881,Z 313.868,A -85,B 0,C 180,E1 -31590,E2 -31590} C_VEL
LIN {X 0,Y 76.261,Z 313.929,A -85,B 0,C 180,E1 -31584.712,E2 -31584.712} C_VEL
LIN {X 0,Y 65.939,Z 313.045,A -85,B 0,C 180,E1 -31573.575,E2 -31573.575} C_VEL
LIN {X 0,Y 60.281,Z 311.529,A -85,B 0,C 180,E1 -31562.203,E2 -31562.203} C_VEL
LIN {X 0,Y 57.522,Z 308.74,A -85,B 0,C 180,E1 -31547.139,E2 -31547.139} C_VEL
LIN {X 0,Y 53.65,Z 310.088,A -85,B 0,C 180,E1 -31549.082,E2 -31549.082} C_VEL
LIN {X 0,Y 48.683,Z 311.893,A -85,B 0,C 180,E1 -31554.729,E2 -31554.729} C_VEL
LIN {X 0,Y 40.727,Z 314.358,A -85,B 0,C 180,E1 -31569.811,E2 -31569.811} C_VEL
LIN {X 0,Y 38.124,Z 314.961,A -85,B 0,C 180,E1 -31579.377,E2 -31579.377} C_VEL
LIN {X 0,Y 36.867,Z 315.13,A -85,B 0,C 180,E1 -31590,E2 -31590} C_VEL
LIN {X 0,Y 38.113,Z 314.962,A -85,B 0,C 180,E1 -31600.626,E2 -31600.626} C_VEL
LIN {X 0,Y 40.726,Z 314.358,A -85,B 0,C 180,E1 -31610.19,E2 -31610.19} C_VEL
LIN {X 0,Y 48.684,Z 311.893,A -85,B 0,C 180,E1 -31625.271,E2 -31625.271} C_VEL
LIN {X 0,Y 53.652,Z 310.088,A -85,B 0,C 180,E1 -31630.917,E2 -31630.917} C_VEL
LIN {X 0,Y 57.487,Z 308.757,A -85,B 0,C 180,E1 -31632.823,E2 -31632.823} C_VEL
LIN {X 0,Y 58.726,Z 310.635,A -85,B 0,C 180,E1 -31623.106,E2 -31623.106} C_VEL
LIN {X 0,Y 61.672,Z 312.106,A -85,B 0,C 180,E1 -31614.272,E2 -31614.272} C_VEL
LIN {X 0,Y 71.319,Z 313.656,A -85,B 0,C 180,E1 -31599.809,E2 -31599.809} C_VEL
LIN {X 0,Y 78.383,Z 313.972,A -85,B 0,C 180,E1 -31593.663,E2 -31593.663} C_VEL
LIN {X 0,Y 78.804,Z 314.009,A -85,B 0,C 180,E1 -31592.694,E2 -31592.694} C_VEL
LIN {X 0,Y 77.936,Z 314.028,A -85,B 0,C 180,E1 -31590.933,E2 -31590.933} C_VEL
LIN {X 0,Y 75.402,Z 314.103,A -85,B 0,C 180,E1 -31588.878,E2 -31588.878} C_VEL
LIN {X 0,Y 64.508,Z 314.141,A -85,B 0,C 180,E1 -31582.513,E2 -31582.513} C_VEL
LIN {X 0,Y 63.375,Z 314.078,A -85,B 0,C 180,E1 -31581.352,E2 -31581.352} C_VEL
LIN {X 0,Y 58.347,Z 313.722,A -85,B 0,C 180,E1 -31574.48,E2 -31574.48} C_VEL
LIN {X 0,Y 53.318,Z 312.59,A -85,B 0,C 180,E1 -31563.404,E2 -31563.404} C_VEL
LIN {X 0,Y 50.748,Z 313.096,A -85,B 0,C 180,E1 -31565.451,E2 -31565.451} C_VEL
LIN {X 0,Y 47.498,Z 314.166,A -85,B 0,C 180,E1 -31572.787,E2 -31572.787} C_VEL
LIN {X 0,Y 45.147,Z 314.77,A -85,B 0,C 180,E1 -31581.044,E2 -31581.044} C_VEL
LIN {X 0,Y 43.963,Z 314.939,A -85,B 0,C 180,E1 -31590,E2 -31590} C_VEL
LIN {X 0,Y 45.138,Z 314.77,A -85,B 0,C 180,E1 -31598.957,E2 -31598.957} C_VEL
LIN {X 0,Y 47.497,Z 314.166,A -85,B 0,C 180,E1 -31607.213,E2 -31607.213} C_VEL
LIN {X 0,Y 50.748,Z 313.096,A -85,B 0,C 180,E1 -31614.549,E2 -31614.549} C_VEL
LIN {X 0,Y 53.319,Z 312.589,A -85,B 0,C 180,E1 -31616.598,E2 -31616.598} C_VEL
LIN {X 0,Y 59.577,Z 313.83,A -85,B 0,C 180,E1 -31603.646,E2 -31603.646} C_VEL
LIN {X 0,Y 70.324,Z 314.233,A -85,B 0,C 180,E1 -31592.12,E2 -31592.12} C_VEL
LIN {X 0,Y 73.176,Z 314.155,A -85,B 0,C 180,E1 -31590,E2 -31590} C_VEL
LIN {X 0,Y 63.375,Z 314.078,A -85,B 0,C 180,E1 -31581.352,E2 -31581.352} C_VEL
LIN {X 0,Y 61.483,Z 314.082,A -85,B 0,C 180,E1 -31580.417,E2 -31580.417} C_VEL
LIN {X 0,Y 58.225,Z 314.244,A -85,B 0,C 180,E1 -31580.689,E2 -31580.689} C_VEL
LIN {X 0,Y 54.62,Z 314.525,A -85,B 0,C 180,E1 -31582.724,E2 -31582.724} C_VEL
LIN {X 0,Y 52.385,Z 314.718,A -85,B 0,C 180,E1 -31585.263,E2 -31585.263} C_VEL
LIN {X 0,Y 51.222,Z 314.717,A -85,B 0,C 180,E1 -31588.553,E2 -31588.553} C_VEL
LIN {X 0,Y 51.086,Z 314.748,A -85,B 0,C 180,E1 -31590,E2 -31590} C_VEL
LIN {X 0,Y 52.204,Z 314.579,A -85,B 0,C 180,E1 -31597.737,E2 -31597.737} C_VEL
LIN {X 0,Y 54.078,Z 314.404,A -85,B 0,C 180,E1 -31599.147,E2 -31599.147} C_VEL
LIN {X 0,Y 62.601,Z 314.439,A -85,B 0,C 180,E1 -31590,E2 -31590} C_VEL
LIN {X 0,Y 54.072,Z 314.405,A -85,B 0,C 180,E1 -31580.869,E2 -31580.869} C_VEL
LIN {X 0,Y 52.213,Z 314.578,A -85,B 0,C 180,E1 -31582.264,E2 -31582.264} C_VEL
LIN {X 0,Y 51.222,Z 314.717,A -85,B 0,C 180,E1 -31588.553,E2 -31588.553} C_VEL
LIN {X 0,Y 51.029,Z 316.716,A -85,B 0,C 180,E1 -31590.73,E2 -31590.73} C_VEL
LIN {X 0,Y 51.029,Z 600,A -85,B 0,C 180,E1 -31590.73,E2 -31590.73} C_VEL
LIN {X 0,Y 51.029,Z 600,A -85,B 0,C 180,E1 -31590.73,E2 -31590.73}

QRS_NEXT_CUT()

QRS_NEXT()
QRS_HOME()

END
